FUNCTION_BLOCK FB_DefGridParamMediator
VAR_INPUT
END_VAR
VAR_OUTPUT
END_VAR
VAR
  _pCreateWorker : POINTER TO FB_WorkerDefGrid_Python;
  _pCamWorker : POINTER TO FB_WorkerDefGrid_Camera;
  _pDefWorker : POINTER TO FB_WorkerDefGrid_Deformation;
  bInitOk     : BOOL;
END_VAR

{attribute 'monitoring':='call'}
PROPERTY fCameraToPrintOffset : LREAL
GET
IF bInitOk THEN
  fCameraToPrintOffset := _pCamWorker^.fCameraToPrintOffset;
END_IF
END_GET
END_PROPERTY

{attribute 'monitoring':='call'}
PROPERTY fDetectToCamera : LREAL
GET
fDetectToCamera := _pCamWorker^.fDetectToCamOffset;
END_GET
END_PROPERTY

METHOD init
VAR_INPUT
  pCreateWorker : POINTER TO FB_WorkerDefGrid_Python;
  pCamWorker : POINTER TO FB_WorkerDefGrid_Camera;
  pDefWorker : POINTER TO FB_WorkerDefGrid_Deformation;
END_VAR
IF pCamWorker <> 0 AND pCamWorker <>0 AND pCreateWorker <> 0 THEN
  _pCreateWorker := pCreateWorker;
  _pCamWorker := pCamWorker;
  _pDefWorker := pDefWorker;
  bInitOk := TRUE;
END_IF
END_METHOD

(*
  Release deformation ct
  TODO: find another way to do inter worker communication for generic methods.
*)
METHOD ReleaseDeformationCT
VAR_INPUT
  iCT              : I_CT;
END_VAR
IF bInitOk THEN
  _pCreateWorker^.DeleteDefCt(iCT:=iCT);
END_IF
END_METHOD

PROPERTY sCameraGridSettings : ST_CameraGridSettings
GET
IF bInitOk THEN
  sCameraGridSettings := _pCamWorker^.sCameraGridSettings;
END_IF
END_GET
END_PROPERTY

PROPERTY sDeformationGridSetttings : ST_DefGridSettings
GET
IF bInitOk THEN
  sDeformationGridSetttings := _pDefWorker^.sDeformationGridSettings;
END_IF
END_GET
END_PROPERTY

END_FUNCTION_BLOCK

(* stored: Version 1.1.0.1, ProductVersion 3.1.4024.3
   POU FB_DefGridParamMediator: Id {9642270e-d441-4770-907b-3f0d0f5dc2e9}, SpecialFunc None
   Property fCameraToPrintOffset: Id {43edb161-94bb-440e-a146-2ecc3ab0b15d}
   Get Get: Id {687dfcbd-6ad8-4ffb-a3c4-66b35289f9de}
   Property fDetectToCamera: Id {0268497d-c5b0-4639-a734-da6955c88aff}
   Get Get: Id {038181c1-f283-429a-835f-ddc555554d78}
   Method init: Id {9cdfcac0-144a-4d88-8e7f-21c6ce0c82c3}
   Method ReleaseDeformationCT: Id {d54eef11-94fc-4211-8079-b54bc203d3ec}
   Property sCameraGridSettings: Id {686354aa-821c-4c68-8c9d-dafadf8ef6fd}
   Get Get: Id {7a8afb02-f662-4c02-aebf-6b3bd22fae1a}
   Property sDeformationGridSetttings: Id {9cf3f096-207d-452b-ace7-3769f0678220}
   Get Get: Id {f92cba8c-0a7c-4567-a017-f6ac55645e3a} *)
